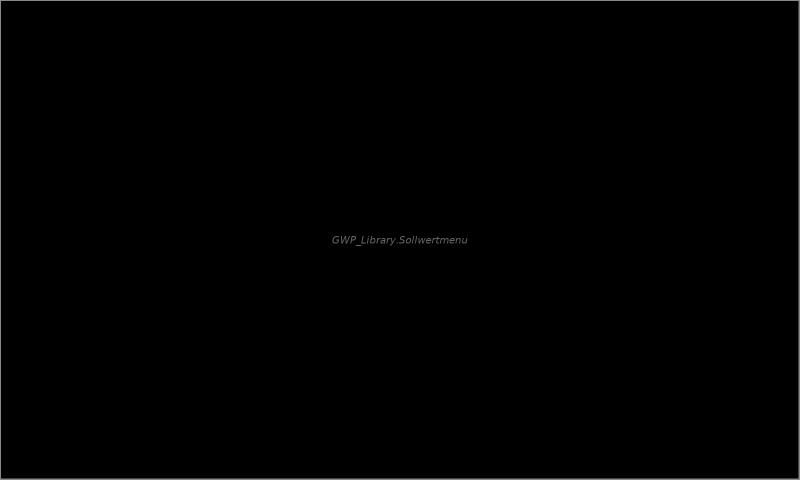
VISUALIZATION Sollwertmenu  // 800x480
    Frame (0,0 800x480)
        shows GWP_Library.Sollwertmenu(FB_Init_1 := Main.Init_0)
END_VISUALIZATION

(* stored: Version 1.1.0.1, ProductVersion 3.1.4022.6
   Visu Sollwertmenu: Id {6dfda5a1-7b2c-400b-a7da-419555e9e987} *)
